FUNCTION_BLOCK DeliveryOrganisation (* Basic Function Block Type *)
  (* Standard: 61499-2 *)
  (* Version 0.0, 11/25/2020, prana, nxtControl GmbH, Template *)
  PACKAGE Main;
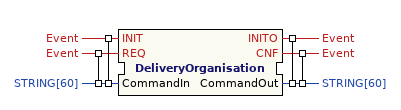
  EVENT_INPUT
    INIT WITH CommandIn; (* Initialization Request *)
    REQ WITH CommandIn; (* Normal Execution Request *)
  END_EVENT
  EVENT_OUTPUT
    INITO WITH CommandOut; (* Initialization Confirm *)
    CNF WITH CommandOut; (* Execution Confirmation *)
  END_EVENT
  VAR_INPUT
    CommandIn : STRING[60]; (* Input event qualifier *)
  END_VAR
  VAR_OUTPUT
    CommandOut : STRING[60]; (* Output event qualifier *)
  END_VAR
  VAR
    i : INT;
    j : INT;
    m : INT;
    n : INT;
    t1 : INT;
    t2 : INT;
    Command : STRING[60];
    m_str : STRING;
  END_VAR
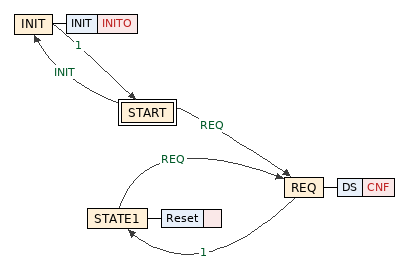
  EC_STATES
    START; (* Initial State *)
    INIT : INIT -> INITO; (* Initialization *)
    REQ : DS -> CNF; (* Normal execution *)
    STATE1 : Reset;
  END_STATES
  EC_TRANSITIONS
    START TO INIT := INIT;
    INIT TO START := 1;
    START TO REQ := REQ;
    REQ TO STATE1 := 1;
    STATE1 TO REQ := REQ;
  END_TRANSITIONS
  ALGORITHM INIT IN ST: (* Initialization algorithm *)
;
  END_ALGORITHM
  ALGORITHM REQ IN ST: (* Normally executed algorithm *)
IF CommandIn = ('C3_to_C5') THEN
	CommandOut := ('C3,P4,D5');
ELSIF CommandIn = ('C5_to_C1') THEN
	CommandOut := ('C5,P6,D1');
ELSIF CommandIn = ('C1_to_C3') THEN
	CommandOut := ('C1,P2,D3');
ELSE
	CommandOut := CommandIn;
END_IF;
  END_ALGORITHM
  ALGORITHM DS IN ST:
i := STRING_TO_INT((RIGHT((LEFT(CommandIn,2)),1)));
j := STRING_TO_INT((RIGHT(CommandIn,1)));

m := i + 1;
n := j-1;
t1 := m;

IF j < i THEN

	FOR t1 := m TO 6 BY 1 DO
		m_str := INT_TO_STRING(m);
		Command := CONCAT(Command,'P',m_str,',');
		m := m + 1;
	END_FOR;

	t1 := 0;

	FOR t1 := 1 TO n BY 1 DO
		m_str := INT_TO_STRING(t1);
		Command := CONCAT(Command,'P',m_str,',');
	END_FOR;

	CommandOut := CONCAT('C',INT_TO_STRING(i),',',Command,'D',INT_TO_STRING(j));


ELSE
	FOR t1 := m TO n BY 1 DO
		m_str := INT_TO_STRING(t1);
		Command := CONCAT(Command,'P',m_str,',');
	END_FOR;
	CommandOut := CONCAT('C',INT_TO_STRING(i),',',Command,'D',INT_TO_STRING(j));

END_IF;
  END_ALGORITHM
  ALGORITHM Reset IN ST:
i := 0;
j := 0;
m := 0;
n := 0;
Command := '';
t1 := 0;
m_str := '';
  END_ALGORITHM
END_FUNCTION_BLOCK
